(* IEC 61131-3 sources: volt/packages/volt-lsp-iec/test-corpus/bakon-nano/Device/Plc Logic/Application/Library Manager/(unresolved)/syssocket interfaces, 17 files *)

(* ---- INADDR.dut ---- *)
TYPE INADDR :
UNION
	S_UN_B : UDINT_IN_BYTES;
	S_UN_W : UDINT_IN_WORDS;
	ULADDR : UDINT;
END_UNION
END_TYPE

(* ---- RTS_SOCKET_SO_VALUE_IP_MREQ.dut ---- *)
TYPE RTS_SOCKET_SO_VALUE_IP_MREQ :
STRUCT
	IMR_MULTIADDR : INADDR;
	IMR_INTERFACE : INADDR;
END_STRUCT
END_TYPE

(* ---- RTS_SOCKET_SO_VALUE_LINGER.dut ---- *)
TYPE RTS_SOCKET_SO_VALUE_LINGER :
STRUCT
	L_ONOFF : WORD;
	L_LINGER : WORD;
END_STRUCT
END_TYPE

(* ---- RTS_SOCKET_SO_VALUE_TCP_KEEPALIVE.dut ---- *)
TYPE RTS_SOCKET_SO_VALUE_TCP_KEEPALIVE :
STRUCT
	BON : DINT;
	PROBES : UDINT;
	PROBESRESULT : RTS_IEC_RESULT;
	TIMEOUT : DINT;
	TIMEOUTRESULT : RTS_IEC_RESULT;
	INTERVAL : DINT;
	INTERVALRESULT : RTS_IEC_RESULT;
END_STRUCT
END_TYPE

(* ---- SOCK_ADAPTER_INFORMATION.dut ---- *)
TYPE SOCK_ADAPTER_INFORMATION :
STRUCT
	UDISTRUCTSIZE : UDINT;
	UDIVERSION : UDINT;
	UDIINDEX : UDINT;
	UDIRESERVED : UDINT;
	WSNAME : WSTRING(ADAPTER_INFO_NAME_LEN);
	WSDESCRIPTION : WSTRING(ADAPTER_INFO_DESC_LEN);
	ABYMAC : ARRAY [0..(ADAPTER_INFO_MAC_ADDR_LENGTH - 1)] OF BYTE;
	WTYPE : WORD;
	DWFLAGS : DWORD;
	IPADDR : INADDR;
	NETMASK : INADDR;
	DEFAULTGATEWAY : INADDR;
END_STRUCT
END_TYPE

(* ---- SOCK_ADAPTER_INFORMATION2.dut ---- *)
TYPE SOCK_ADAPTER_INFORMATION2 :
STRUCT
	UDISTRUCTSIZE : UDINT;
	UDIVERSION : UDINT;
	UDIINDEX : UDINT;
	UDIRESERVED : UDINT;
	WSNAME : WSTRING(ADAPTER_INFO_NAME_LEN);
	WSDESCRIPTION : WSTRING(ADAPTER_INFO_DESC_LEN);
	ABYMAC : ARRAY [0..(ADAPTER_INFO_MAC_ADDR_LENGTH - 1)] OF BYTE;
	WTYPE : WORD;
	DWFLAGS : DWORD;
	IPADDR : INADDR;
	NETMASK : INADDR;
	DEFAULTGATEWAY : INADDR;
	PRIMARYNAMESERVER : INADDR;
	SECONDARYNAMESERVER : INADDR;
	WSDNSSUFFIX : WSTRING(ADAPTER_INFO_DNSSUFFIX_LEN);
	DHCPSERVER : INADDR;
END_STRUCT
END_TYPE

(* ---- SOCK_ADAPTER_INFORMATION3.dut ---- *)
TYPE SOCK_ADAPTER_INFORMATION3 :
STRUCT
	UDISTRUCTSIZE : UDINT;
	UDIVERSION : UDINT;
	UDIINDEX : UDINT;
	UDIRESERVED : UDINT;
	WSNAME : WSTRING(ADAPTER_INFO_NAME_LEN);
	WSDESCRIPTION : WSTRING(ADAPTER_INFO_DESC_LEN);
	ABYMAC : ARRAY [0..(ADAPTER_INFO_MAC_ADDR_LENGTH - 1)] OF BYTE;
	WTYPE : WORD;
	DWFLAGS : DWORD;
	IPADDR : INADDR;
	NETMASK : INADDR;
	DEFAULTGATEWAY : INADDR;
	PRIMARYNAMESERVER : INADDR;
	SECONDARYNAMESERVER : INADDR;
	WSDNSSUFFIX : WSTRING(ADAPTER_INFO_DNSSUFFIX_LEN);
	DHCPSERVER : INADDR;
	UDIOSINDEX : UDINT;
END_STRUCT
END_TYPE

(* ---- SOCK_HOSTENT.dut ---- *)
TYPE SOCK_HOSTENT :
STRUCT
	SZHOSTNAME : REFERENCE TO STRING;
	PALIASLIST : POINTER TO POINTER TO STRING;
	IHOSTADDRTYPE : INT;
	ILENGTHADDR : INT;
	PADDRLIST : POINTER TO POINTER TO STRING;
END_STRUCT
END_TYPE

(* ---- SOCK_RECVMSG_MSG.dut ---- *)
TYPE SOCK_RECVMSG_MSG :
STRUCT
	PBUFFER : POINTER TO BYTE;
	LENGTH : __XWORD;
	ADDRESS : SOCKADDRESS;
	MSGFLAGS : DWORD;
	MSGFLAGSSUPPORTED : DWORD;
END_STRUCT
END_TYPE

(* ---- SOCKADDRESS.dut ---- *)
TYPE SOCKADDRESS :
STRUCT
	SIN_FAMILY : INT;
	SIN_PORT : UINT;
	SIN_ADDR : INADDR;
	SIN_ZERO : ARRAY [0..7] OF BYTE;
END_STRUCT
END_TYPE

(* ---- SOCKET_FD_SET.dut ---- *)
TYPE SOCKET_FD_SET :
STRUCT
	FD_COUNT : UDINT;
	FD_ARRAY : ARRAY [0..(SOCKET_FD_SETSIZE - 1)] OF RTS_IEC_HANDLE;
END_STRUCT
END_TYPE

(* ---- SOCKET_TIMEVAL.dut ---- *)
TYPE SOCKET_TIMEVAL :
STRUCT
	TV_SEC : DINT;
	TV_USEC : DINT;
END_STRUCT
END_TYPE

(* ---- UDINT_IN_BYTES.dut ---- *)
TYPE UDINT_IN_BYTES :
STRUCT
	S_B1 : BYTE;
	S_B2 : BYTE;
	S_B3 : BYTE;
	S_B4 : BYTE;
END_STRUCT
END_TYPE

(* ---- UDINT_IN_WORDS.dut ---- *)
TYPE UDINT_IN_WORDS :
STRUCT
	S_W1 : WORD;
	S_W2 : WORD;
END_STRUCT
END_TYPE

(* ---- UDP_REPLY.dut ---- *)
TYPE UDP_REPLY :
STRUCT
	ULSOURCEADDRESS : UDINT;
	SZSOURCEADDRESS : STRING(29);
	DIRECV : __XINT;
END_STRUCT
END_TYPE

(* ---- UDP_REPLY2.dut ---- *)
TYPE UDP_REPLY2 :
STRUCT
	ULSOURCEADDRESS : UDINT;
	SZSOURCEADDRESS : STRING(31);
	DIRECV : __XINT;
	USRECVPORT : WORD;
END_STRUCT
END_TYPE

(* ---- GVL.gvl ---- *)
VAR_GLOBAL
	SOCKET_AF_UNSPEC : INT := 0;
	SOCKET_AF_LOCAL : INT := 1;
	SOCKET_AF_UNIX : INT := 1;
	SOCKET_AF_INET : INT := 2;
	SOCKET_AF_IMPLINK : INT := 3;
	SOCKET_AF_PUP : INT := 4;
	SOCKET_AF_CHAOS : INT := 5;
	SOCKET_AF_NS : INT := 6;
	SOCKET_AF_ISO : INT := 7;
	SOCKET_AF_OSI : INT := 7;
	SOCKET_AF_ECMA : INT := 8;
	SOCKET_AF_DATAKIT : INT := 9;
	SOCKET_AF_CCITT : INT := 10;
	SOCKET_AF_SNA : INT := 11;
	SOCKET_AF_DECNET : INT := 12;
	SOCKET_AF_DLI : INT := 13;
	SOCKET_AF_LAT : INT := 14;
	SOCKET_AF_HYLINK : INT := 15;
	SOCKET_AF_APPLETALK : INT := 16;
	SOCKET_AF_ROUTE : INT := 17;
	SOCKET_AF_LINK : INT := 18;
	SOCKET_PSEUDO_AF_XTP : INT := 19;
	SOCKET_AF_COIP : INT := 20;
	SOCKET_AF_CNT : INT := 21;
	SOCKET_PSEUDO_AF_RTIP : INT := 22;
	SOCKET_AF_IPX : INT := 23;
	SOCKET_AF_SIP : INT := 24;
	SOCKET_PSEUDO_AF_PIP : INT := 25;
	SOCKET_AF_MAX : INT := 26;
	SOCKET_AF_INET_BSD : INT := 100;
	SOCKET_AF_INET_STREAMS : INT := 101;
	SOCKET_IPPROTO_IP : DINT := 0;
	SOCKET_IPPROTO_ICMP : DINT := 1;
	SOCKET_IPPROTO_IGMP : DINT := 2;
	SOCKET_IPPROTO_GGP : DINT := 3;
	SOCKET_IPPROTO_TCP : DINT := 6;
	SOCKET_IPPROTO_PUP : DINT := 12;
	SOCKET_IPPROTO_UDP : DINT := 17;
	SOCKET_IPPROTO_IDP : DINT := 22;
	SOCKET_IPPROTO_ND : DINT := 77;
	SOCKET_IPPROTO_TLS : DINT := 254;
	SOCKET_IPPROTO_RAW : DINT := 255;
	SOCKET_IPPROTO_MAX : DINT := 256;
	SOCKET_SOL : DINT := 16#FFFF;
	SOCKET_DEVICE_SPECIFIC : DINT := ANY_TO_DINT(16#80000000);
	SOCKET_SO_DEBUG : DINT := 16#1;
	SOCKET_SO_ACCEPTCONN : DINT := 16#2;
	SOCKET_SO_REUSEADDR : DINT := 16#4;
	SOCKET_SO_KEEPALIVE : DINT := 16#8;
	SOCKET_SO_DONTROUTE : DINT := 16#10;
	SOCKET_SO_BROADCAST : DINT := 16#20;
	SOCKET_SO_USELOOPBACK : DINT := 16#40;
	SOCKET_SO_LINGER : DINT := 16#80;
	SOCKET_SO_OOBINLINE : DINT := 16#100;
	SOCKET_SO_REUSEPORT : DINT := 16#200;
	SOCKET_SO_SNDBUF : DINT := 16#1001;
	SOCKET_SO_RCVBUF : DINT := 16#1002;
	SOCKET_SO_SNDLOWAT : DINT := 16#1003;
	SOCKET_SO_RCVLOWAT : DINT := 16#1004;
	SOCKET_SO_SNDTIMEO : DINT := 16#1005;
	SOCKET_SO_RCVTIMEO : DINT := 16#1006;
	SOCKET_SO_ERROR : DINT := 16#1007;
	SOCKET_SO_TYPE : DINT := 16#1008;
	SOCKET_SO_PROTOTYPE : DINT := 16#1009;
	SOCKET_SO_HOSTNAME : DINT := 16#2001;
	SOCKET_SO_STARTTLS : DINT := 16#3001;
	SOCKET_TCP_NODELAY : DINT := 16#1;
	SOCKET_TCP_MAXSEG : DINT := 16#2;
	SOCKET_IP_TOS : DINT := 16#1;
	SOCKET_IP_MULTICAST_IF : DINT := 16#9;
	SOCKET_SO_MULTICAST_IF : DINT := 16#9;
	SOCKET_IP_MULTICAST_TTL : DINT := 16#A;
	SOCKET_IP_MULTICAST_LOOP : DINT := 16#B;
	SOCKET_IP_ADD_MEMBERSHIP : DINT := 16#C;
	SOCKET_IP_DROP_MEMBERSHIP : DINT := 16#D;
	SOCKET_IP_DONTFRAGMENT : DINT := 16#E;
	SOCKET_IP_PKTINFO : DINT := 16#13;
	SOCKET_STREAM : DINT := 1;
	SOCKET_DGRAM : DINT := 2;
	SOCKET_RAW : DINT := 3;
	SOCKET_RDM : DINT := 4;
	SOCKET_SEQPACKET : DINT := 5;
	SOCKET_INADDR_ANY : UDINT := 16#0;
	SOCKET_INADDR_LOOPBACK : UDINT := 16#7F000001;
	SOCKET_INADDR_BROADCAST : UDINT := 16#FFFFFFFF;
	SOCKET_INADDR_NONE : UDINT := 16#FFFFFFFF;
	SOCKET_FIONREAD : DINT := 1;
	SOCKET_FIONBIO : DINT := 2;
	SOCKET_MSG_NONE : DINT := 16#0;
	SOCKET_MSG_OOB : DINT := 16#1;
	SOCKET_MSG_PEEK : DINT := 16#2;
	SOCKET_MSG_DONTROUTE : DINT := 16#4;
	SOCKET_MSG_DONTWAIT : DINT := 16#8;
	SOCKET_MSG_BCAST : DINT := 16#400;
	SOCKET_MSG_MCAST : DINT := 16#800;
	SOCKET_SD_RECEIVE : DINT := 16#0;
	SOCKET_SD_SEND : DINT := 16#1;
	SOCKET_SD_BOTH : DINT := 16#2;
	SOCKET_FD_SETSIZE : DINT := 64;
	MAX_SOCKET_FD_SETSIZE : DINT := 63;
	ADAPTER_INFO_MAC_ADDR_LENGTH : INT := 6;
	ADAPTER_INFO_NAME_LEN : INT := 255;
	ADAPTER_INFO_DESC_LEN : INT := 255;
	ADAPTER_INFO_DNSSUFFIX_LEN : INT := 255;
	SOCK_AIT_ETHERNET : WORD := 1;
	SOCK_AIT_LOCALHOST : WORD := 2;
	SOCK_AIT_PPP : WORD := 3;
	SOCK_AIT_WIRELESS : WORD := 4;
	SOCK_AIF_NONE : DWORD := 16#0;
	SOCK_AIF_INACTIVE : DWORD := 16#1;
	SOCK_AIF_ALIAS_IP : DWORD := 16#2;
	SOCK_AIF_DYNAMIC_IP : DWORD := 16#4;
	SOCK_AIF_FIX_IP : DWORD := 16#8;
	SOCK_AIF_IP_CHANGE_ALLOWED : DWORD := 16#10;
	SOCK_AIF_GATEWAY_INFO_VALID : DWORD := 16#20;
	SOCK_AIF_DNS_INFO_VALID : DWORD := 16#40;
	SOCK_AIF_DHCP_INFO_VALID : DWORD := 16#80;
	SOCK_AIF_INFO_VALID : DWORD := 16#8000;
END_VAR
